TYPE ST_System_HES_Zustand :
STRUCT
	Betrieb_Anford			: BOOL;
	Betrieb_Soll				: BOOL;
	Betrieb					: BOOL;

	Netze_Anford				: ST_Zustand_Netze_Anford;

	Freigabe					: BOOL;
	Freigabe_Deakt			: BOOL;
	Freigabe_Code			: WORD;

	Stoerung					: BOOL;
	Stoerung_Code			: WORD;

	Warnung					: BOOL;
	Warnung_Code			: WORD;

	Status					: SINT;
	Status_Vorl_Stellventil		: BOOL;
	Status_Vorl_Pumpe		: BOOL;
	Status_Nachl_Stellventil	: BOOL;
	Status_Nachl_Pumpe		: BOOL;

	Quittierung				: BOOL;

	Netz_KW_Anford			: ST_Zustand_Netz_Anford; (* Philipp *)

END_STRUCT
END_TYPE

(* stored: Version 1.1.0.1, ProductVersion 3.1.4024.9
   DUT ST_System_HES_Zustand: Id {20c3bc31-e742-4e2a-9d89-11be46d7bead} *)
